FUNCTION_BLOCK FB_Gantry
VAR_INPUT
	bExecuteHeatSetCycle 	: BOOL;
	bGoHome 				: BOOL;
	bGoPreHeatSet 			: BOOL;
	bGoHeatSet 				: BOOL;
	bGoPreQuench 			: BOOL;
	bGoQuench 				: BOOL;
END_VAR
VAR_OUTPUT
	bAtHome 				: BOOL;
	bAtPreHeatSet 			: BOOL;
	bAtHeatSet 				: BOOL;
	bAtPreQuench 			: BOOL;
	bAtQuench 				: BOOL;
END_VAR
VAR
	IpAddrX : STRING(15) := '10.10.10.1';
	IpAddrZ : STRING(15) := '10.10.10.2';
	TcpPort : INT := 502;
	nUnitID : BYTE := 255;
END_VAR

METHOD M_HeatSoak : BOOL
VAR_INPUT
END_VAR
END_METHOD

METHOD M_Home : BOOL
VAR_INPUT
END_VAR
END_METHOD

METHOD M_Quench : BOOL
VAR_INPUT
END_VAR
END_METHOD

END_FUNCTION_BLOCK

(* stored: Version 1.1.0.1, ProductVersion 3.1.4024.10
   POU FB_Gantry: Id {b7979926-7c32-4a40-91b9-f80b9f875b86}, SpecialFunc None
   Method M_HeatSoak: Id {19339519-3588-48a6-b846-72bfab32be0d}
   Method M_Home: Id {1e0502fa-b362-416e-8dd0-a04418b7d6ba}
   Method M_Quench: Id {8ac75d54-3dc9-4695-a395-72b1be965303} *)
